PROGRAM interlocks
VAR PERSISTENT
END_VAR

// NETWORK 1

END_PROGRAM

(* stored: Version 1.1.0.1, ProductVersion 3.1.4024.12
   POU interlocks: Id {5e6ac187-5fbb-479f-b495-0ce9f8a80e37}, SpecialFunc None *)
